% RSLogix 500 project 08-TRAFFICLIGHTSDELUXETWOWAY_BAK077.RSS, saved by version 9.00.00.04 %
PROJECT "UNTITLED"    % processor: MicroLogix 1200 %

PROGRAM FILES
  LAD 2 "MAIN_PROG"  12 rungs
  LAD 3 "USER_FAULT"  1 rungs
  LAD 4 "HSC_INT"  1 rungs
  LAD 5 "STI_INT"  1 rungs
  LAD 6, 7, 8, 9, 10, 11, 12, 13, 14, 15, 16: only END

DATA FILES
  O0 OUTPUT  4 elements
  I1 INPUT  4 elements
  S2 STATUS  66 elements
  B3 BINARY  32 elements
  T4 TIMER  40 elements
  C5 COUNTER  32 elements
  R6 CONTROL  16 elements
  N7 INTEGER  105 elements
  F8 FLOAT  1 elements

LADDER 2 "MAIN_PROG"
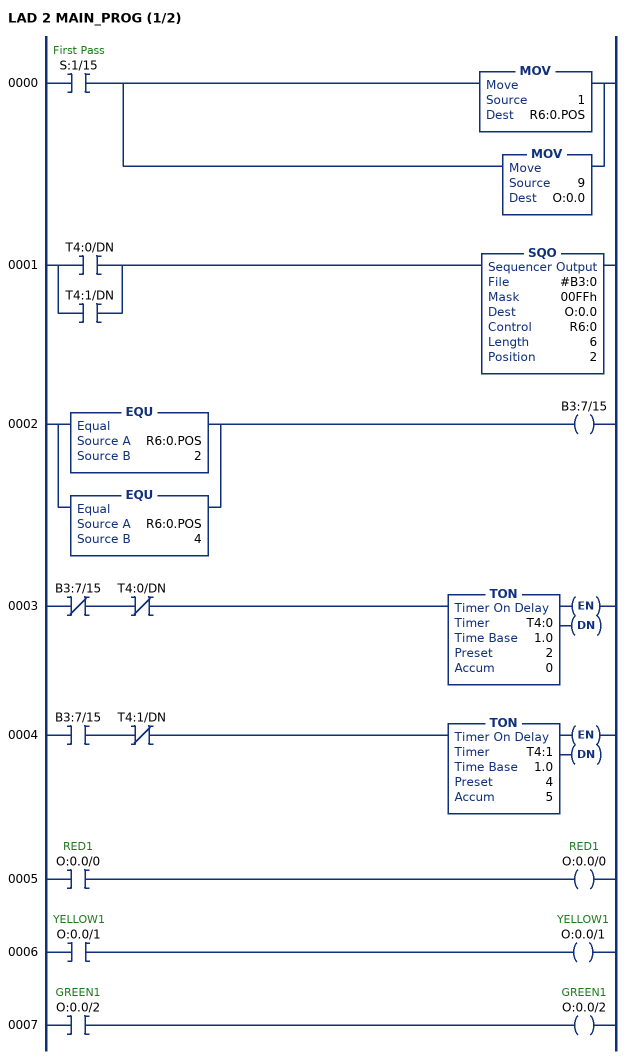
% Rung: 0 %
SOR XIC S:1/15 BST MOV 1 R6:0.POS NXB MOV 9 O:0.0 BND EOR
%   S:1/15  "First Pass" %
% Rung: 1 %
SOR BST XIC T4:0/DN NXB XIC T4:1/DN BND SQO #B3:0 00FFh O:0.0 R6:0 6 2 EOR
% Rung: 2 %
SOR BST EQU R6:0.POS 2 NXB EQU R6:0.POS 4 BND OTE B3:7/15 EOR
% Rung: 3 %
SOR XIO B3:7/15 XIO T4:0/DN TON T4:0 1.0 2 0 EOR
% Rung: 4 %
SOR XIC B3:7/15 XIO T4:1/DN TON T4:1 1.0 4 5 EOR
% Rung: 5 %
SOR XIC O:0.0/0 OTE O:0.0/0 EOR
%   O:0.0/0  "RED1" %
% Rung: 6 %
SOR XIC O:0.0/1 OTE O:0.0/1 EOR
%   O:0.0/1  "YELLOW1" %
% Rung: 7 %
SOR XIC O:0.0/2 OTE O:0.0/2 EOR
%   O:0.0/2  "GREEN1" %

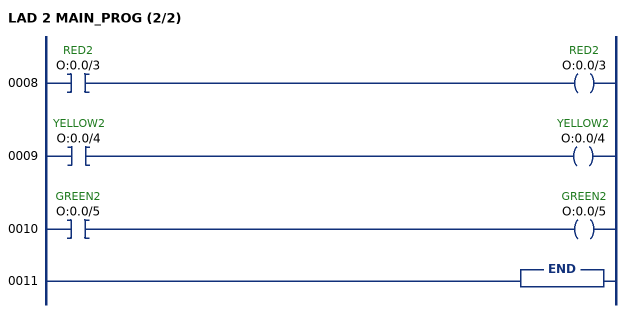
% Rung: 8 %
SOR XIC O:0.0/3 OTE O:0.0/3 EOR
%   O:0.0/3  "RED2" %
% Rung: 9 %
SOR XIC O:0.0/4 OTE O:0.0/4 EOR
%   O:0.0/4  "YELLOW2" %
% Rung: 10 %
SOR XIC O:0.0/5 OTE O:0.0/5 EOR
%   O:0.0/5  "GREEN2" %
% Rung: 11 %
SOR END EOR

OTHER DOCUMENTED ADDRESSES
  RED1  

DATA TABLE (non-zero values as saved)
DATA B3
% B3:0 % 0X0000 0X0009 0X000C 0X000A 0X0009 0X0021 0X0011 0X0000 0X0000 0X0000
DATA T4
% .PRE .ACC %
% T4:0 % 2 0
% T4:1 % 4 5
DATA R6
% .LEN .POS %
% R6:0 % 6 2
